PROGRAM SLTC_EXTRA
VAR
END_VAR

END_PROGRAM

(* stored: Version 1.1.0.1, ProductVersion 3.1.4022.18
   POU SLTC_EXTRA: Id {81772848-36a2-43b7-b61c-16cc38a214e2}, SpecialFunc None *)
